FUNCTION_BLOCK FB_Mediator IMPLEMENTS I_Mediator
VAR_INPUT
	iColleague : ARRAY [1..Param.MAX_COLLEAGUES] OF I_Colleague; // Colleague Interface Array
END_VAR

METHOD notify : BOOL
VAR_INPUT
	(* Colleague sending the notification*)
	sender	: I_Colleague;
	(* Some event the collegue is attempting*)
	event	: STRING;
END_VAR

VAR
	i: INT;
END_VAR
FOR i := 1 TO Param.MAX_COLLEAGUES DO
		IF iColleague[i] <> 0 AND iColleague[i] = sender THEN
			ADSLOGSTR(msgCtrlMask := ADSLOG_MSGTYPE_MSGBOX, msgFmtStr := CONCAT(CONCAT('User ', TO_STRING(i)), ' said: %s'), strArg := event);
		END_IF
END_FOR
END_METHOD

END_FUNCTION_BLOCK

(* stored: Version 1.1.0.1, ProductVersion 3.1.4024.12
   POU FB_Mediator: Id {9da9c772-232d-4988-8017-ee328e3fdbeb}, SpecialFunc None
   Method notify: Id {c2bd4c05-5ba7-41fe-928b-db76afe4fa0e} *)
